Staubli VAL3: onStart.pgx

public program onStart(string& x_sItem[])
  local num i
  local string l_sType
begin
// on START
end
